INTERFACE ITF_TopElement2 EXTENDS ITF_BaseTopElement

END_INTERFACE

(* stored: Version 1.1.0.1
   Itf ITF_TopElement2: Id {a9f8ec62-a8bb-0704-3758-0ada0ec161eb} *)
